// TIA Portal V20 export
DATA_BLOCK "TASK"   // DB41
{ S7_Optimized_Access := 'FALSE' }
VERSION : 0.1
// stored: AutoNumber true, DBAccessibleFromOPCUA true, DBAccessibleFromWebserver true, IsOnlyStoredInLoadMemory false, IsWriteProtectedInAS false
   VAR RETAIN
      Status { ExternalWritable := 'False'} : "LGR_Equip_TaskStatus";
      Proc { ExternalWritable := 'False'} : "LGR_Proc_component";
      ProcBuff { ExternalWritable := 'False'} : "LGR_Proc_component";
      Now { ExternalWritable := 'False'} : "LGR_Task_Data";
      NowBuff { S7_SetPoint := 'True'} : "LGR_Task_Data";
      Buff { ExternalWritable := 'False'} : Array[0..3] of "LGR_Task_Data";
      Last { ExternalWritable := 'False'} : Array[0..9] of "LGR_Task_Data";
      Canceled { S7_SetPoint := 'True'} : Array[0..9] of "LGR_Task_Data";
      Rejected { S7_SetPoint := 'True'} : Array[0..9] of "LGR_Task_Data";
      ErrorOccuredData : Struct
         Last { S7_SetPoint := 'True'} : Array[0..9] of "LGR_Task_Data";
         Now { S7_SetPoint := 'True'} : Array[0..9] of "LGR_Task_Data";
         Next { S7_SetPoint := 'True'} : Array[0..9] of "LGR_Task_Data";
         "Time" { S7_SetPoint := 'True'} : Array[0..9] of DTL;
      END_STRUCT;
   END_VAR
BEGIN
END_DATA_BLOCK
